FUNCTION TryConvert_UINT_TO_INT : BOOL
VAR_INPUT
	in : UINT;
	out : REFERENCE TO INT;
END_VAR

IF in > DatatypeLimits.MAX_VALUE_OF_UINT_WHICH_CAN_BE_HELD_IN_A_INT THEN
	RETURN;
END_IF

out := UINT_TO_INT(in);
TryConvert_UINT_TO_INT := TRUE;

END_FUNCTION

(* stored: Version 1.1.0.1, ProductVersion 3.1.4024.12
   POU TryConvert_UINT_TO_INT: Id {7a1dea8d-834c-4fc8-bf0a-d44e944852b0}, SpecialFunc None *)
